FUNCTION_BLOCK Switches
  (* Standard: 61499-2 *)
  (* Version 0.1, 2017-00-17, hpea485, UOA *)
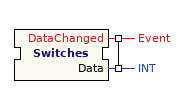
  EVENT_OUTPUT
    DataChanged WITH Data;
  END_EVENT
  VAR_OUTPUT
    Data : INT;
  END_VAR
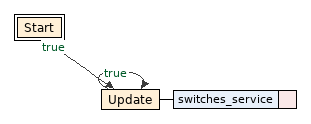
  EC_STATES
    Start;
    Update : switches_service;
  END_STATES
  EC_TRANSITIONS
    Start TO Update := true;
    Update TO Update := true;
  END_TRANSITIONS
  ALGORITHM switches_service IN C:
if(SWITCHES != me->Data) {
	me->Data = SWITCHES;
	me->outputEvents.event.DataChanged = 1;
}
  END_ALGORITHM
END_FUNCTION_BLOCK
